{attribute 'GeneratedUsingTerminal: EK1122-0000-0018'}
{attribute addProperty BoxType "EK1122-0000-0018"}
{attribute addProperty Id "Beckhoff_BKxxxxsub_EK1100Beckhoff_BKxxxxsub_EK1100_59A469240A_0001_BK1120_0000_0000A_0001_BK1120_0000_0000_205E65590A_0002_BK1120_0000_0001A_0002_BK1120_0000_0001_76F1F8EB0A_0003_BK1120_0000_0016A_0003_BK1120_0000_0016_8D015E3D0A_0004_BK1120_0000_0017A_0004_BK1120_0000_0017_DBAEC38F0A_0005_BK1120_0000_0018A_0005_BK1120_0000_0018_C2DFD8D80A_0006_BK1120_0000_0019A_0006_BK1120_0000_0019_9470456A0A_0007_BK1120_0000_0020A_0007_BK1120_0000_0020_61E272590A_0008_BK1120_0000_0021A_0008_BK1120_0000_0021_374DEFEB0A_0009_CPXXXX_BK1150_0016A_0009_CPXXXX_BK1150_0016_CCBD493D0A_0010_BK1150_0000_0016A_0010_BK1150_0000_0016_9A12D48F0A_0011_BK1150_0000_0017A_0011_BK1150_0000_0017_3F9D19260A_0012_BK1150_0000_0018A_0012_BK1150_0000_0018_693284940A_0013_BK1150_0000_0019A_0013_BK1150_0000_0019_92C222420Term_19_EK1100Term_19_EK1100_718FBBA40Term_23_EK1100Term_23_EK1100_08A82DAA0Term_21_EK1100Term_21_EK1100_FD75FF180A_0019_IL2300_B110_0016A_0019_IL2300_B110_0016_AC908CDE0A_0020_IL2300_B110_0017A_0020_IL2300_B110_0017_8C062E240A_0021_IL2301_B110_0016A_0021_IL2301_B110_0016_FF61810D0A_0022_IL2301_B110_0017A_0022_IL2301_B110_0017_BAC34F2E0A_0023_IL2302_B110_0016A_0023_IL2302_B110_0016_19AEDF5F0A_0024_IL2302_B110_0017A_0024_IL2302_B110_0017_E18CEC300"}
{attribute addProperty CRC "3274467932"}
{attribute addProperty Size "0"}
TYPE Beckhoff_BKxxxxEK1122_C32C6A5C EXTENDS EK1122_1FC0878B :
STRUCT
	{attribute addProperty Name "Beckhoff_BKxxxxsub_EK1100"}
	Beckhoff_BKxxxxsub_EK1100 : Beckhoff_BKxxxxsub_EK1100_59A46924;
	{attribute addProperty Name "A_0001_BK1120_0000_0000"}
	A_0001_BK1120_0000_0000 : A_0001_BK1120_0000_0000_205E6559;
	{attribute addProperty Name "A_0002_BK1120_0000_0001"}
	A_0002_BK1120_0000_0001 : A_0002_BK1120_0000_0001_76F1F8EB;
	{attribute addProperty Name "A_0003_BK1120_0000_0016"}
	A_0003_BK1120_0000_0016 : A_0003_BK1120_0000_0016_8D015E3D;
	{attribute addProperty Name "A_0004_BK1120_0000_0017"}
	A_0004_BK1120_0000_0017 : A_0004_BK1120_0000_0017_DBAEC38F;
	{attribute addProperty Name "A_0005_BK1120_0000_0018"}
	A_0005_BK1120_0000_0018 : A_0005_BK1120_0000_0018_C2DFD8D8;
	{attribute addProperty Name "A_0006_BK1120_0000_0019"}
	A_0006_BK1120_0000_0019 : A_0006_BK1120_0000_0019_9470456A;
	{attribute addProperty Name "A_0007_BK1120_0000_0020"}
	A_0007_BK1120_0000_0020 : A_0007_BK1120_0000_0020_61E27259;
	{attribute addProperty Name "A_0008_BK1120_0000_0021"}
	A_0008_BK1120_0000_0021 : A_0008_BK1120_0000_0021_374DEFEB;
	{attribute addProperty Name "A_0009_CPXXXX_BK1150_0016"}
	A_0009_CPXXXX_BK1150_0016 : A_0009_CPXXXX_BK1150_0016_CCBD493D;
	{attribute addProperty Name "A_0010_BK1150_0000_0016"}
	A_0010_BK1150_0000_0016 : A_0010_BK1150_0000_0016_9A12D48F;
	{attribute addProperty Name "A_0011_BK1150_0000_0017"}
	A_0011_BK1150_0000_0017 : A_0011_BK1150_0000_0017_3F9D1926;
	{attribute addProperty Name "A_0012_BK1150_0000_0018"}
	A_0012_BK1150_0000_0018 : A_0012_BK1150_0000_0018_69328494;
	{attribute addProperty Name "A_0013_BK1150_0000_0019"}
	A_0013_BK1150_0000_0019 : A_0013_BK1150_0000_0019_92C22242;
	{attribute addProperty Name "Term_19_EK1100"}
	Term_19_EK1100 : Term_19_EK1100_718FBBA4;
	{attribute addProperty Name "Term_23_EK1100"}
	Term_23_EK1100 : Term_23_EK1100_08A82DAA;
	{attribute addProperty Name "Term_21_EK1100"}
	Term_21_EK1100 : Term_21_EK1100_FD75FF18;
	{attribute addProperty Name "A_0019_IL2300_B110_0016"}
	A_0019_IL2300_B110_0016 : A_0019_IL2300_B110_0016_AC908CDE;
	{attribute addProperty Name "A_0020_IL2300_B110_0017"}
	A_0020_IL2300_B110_0017 : A_0020_IL2300_B110_0017_8C062E24;
	{attribute addProperty Name "A_0021_IL2301_B110_0016"}
	A_0021_IL2301_B110_0016 : A_0021_IL2301_B110_0016_FF61810D;
	{attribute addProperty Name "A_0022_IL2301_B110_0017"}
	A_0022_IL2301_B110_0017 : A_0022_IL2301_B110_0017_BAC34F2E;
	{attribute addProperty Name "A_0023_IL2302_B110_0016"}
	A_0023_IL2302_B110_0016 : A_0023_IL2302_B110_0016_19AEDF5F;
	{attribute addProperty Name "A_0024_IL2302_B110_0017"}
	A_0024_IL2302_B110_0017 : A_0024_IL2302_B110_0017_E18CEC30;
END_STRUCT
END_TYPE

(* stored: Version 1.2.0.0, ProductVersion 3.1.4024.9
   DUT Beckhoff_BKxxxxEK1122_C32C6A5C: Id {7f3e8d9c-3520-4c30-be29-0087a53a1fcb} *)
